Staubli VAL3: motionProgress.pgx

public program motionProgress(num x_nMoveId, num x_nMotProg)
begin

  // display nMoveId and nMotionProgress

  userPageSet("uxMonitor", "lblMoveId", "innerHTML", x_nMoveId)
  userPageSet("uxMonitor", "lblMotionProgress", "innerHTML", x_nMotProg)

end
